(* PLC project SafeLOGIC, BrAutomation SafeDESIGNER  5.24.1.0 *)
(* stored: companyURL http://www.br-automation.com, creationDateTime Sun Oct 26 13:09:37 2025 *)

PROGRAM HeatWater

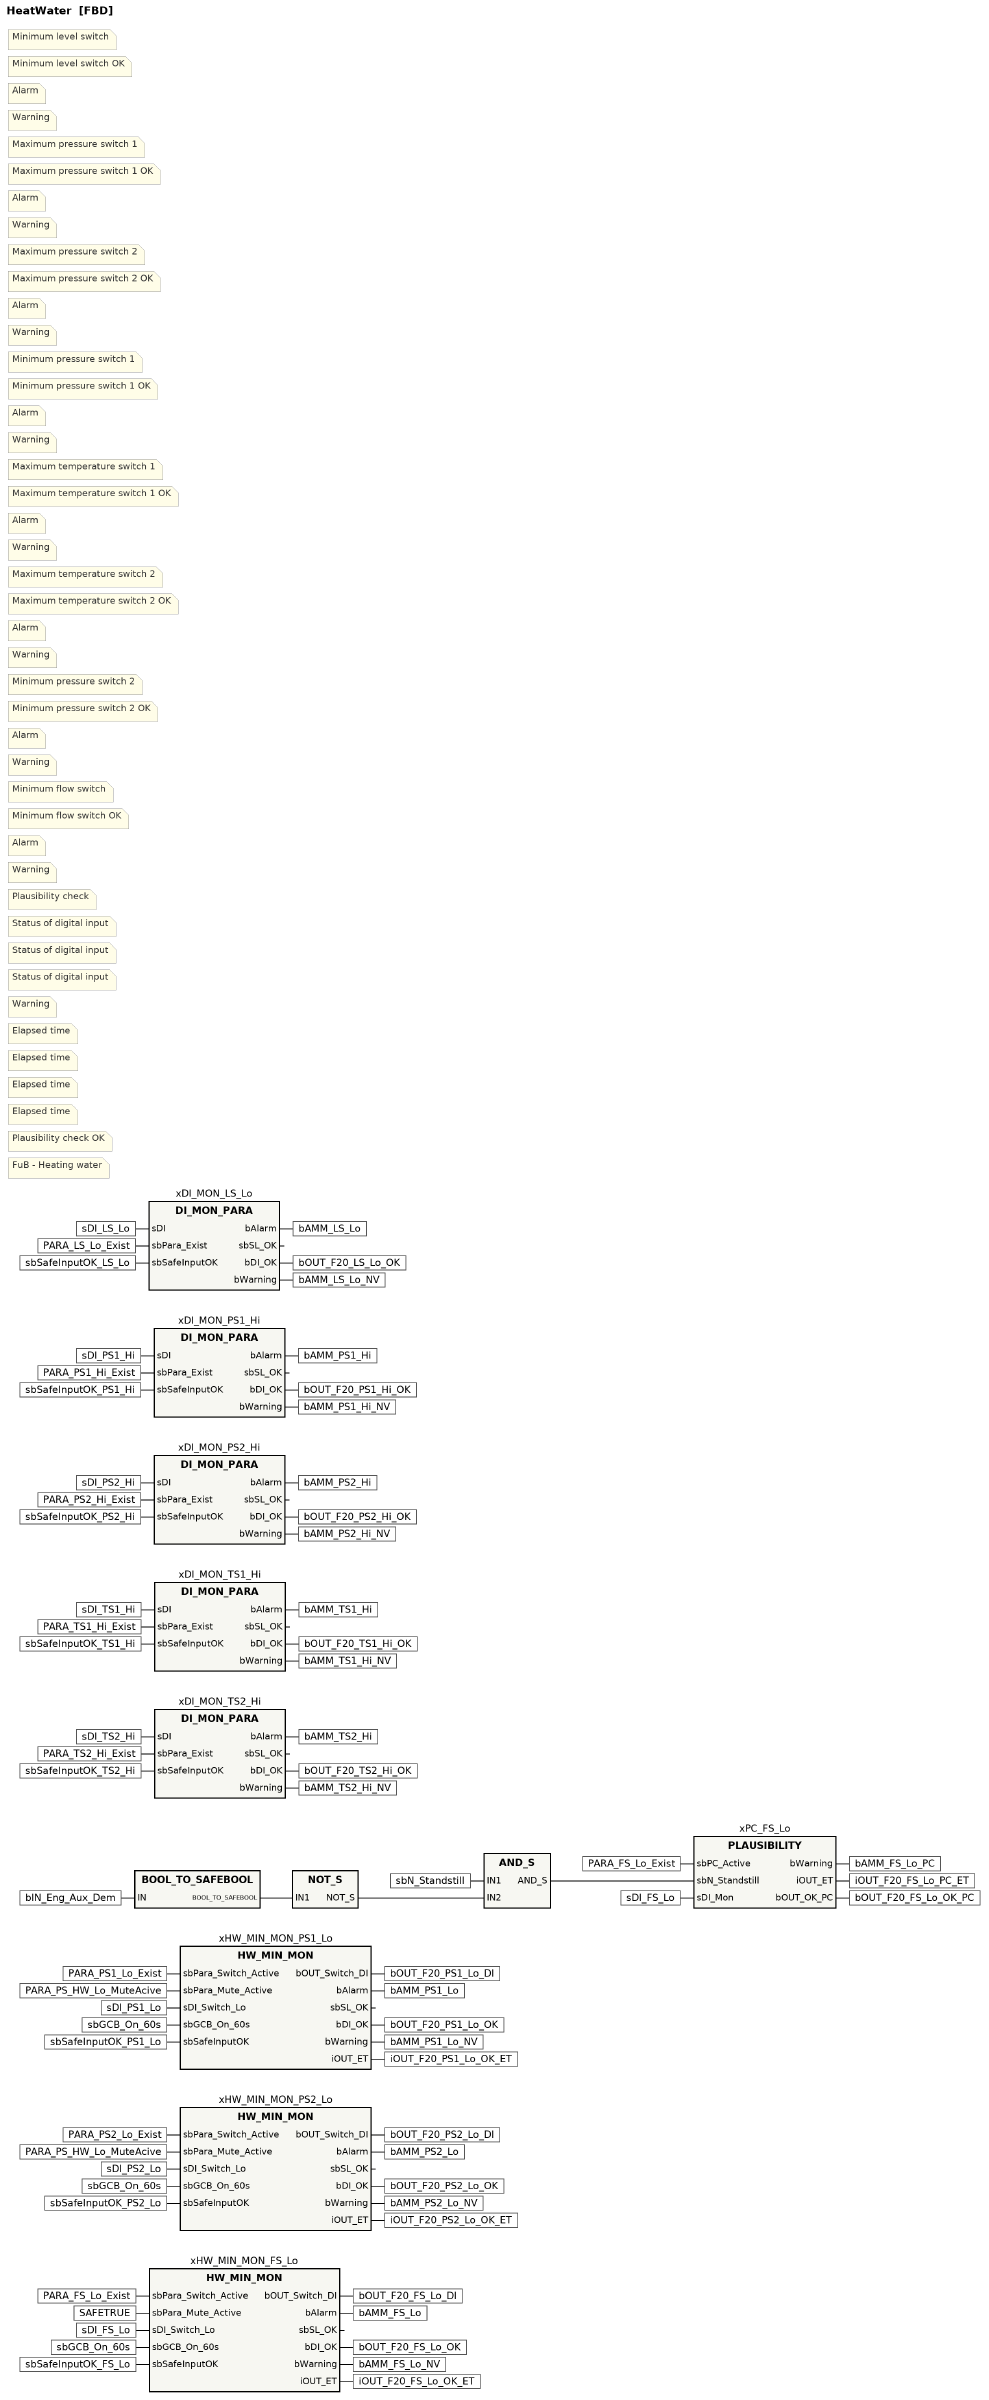
(* FBD diagram, written out as Structured Text *)
(* FuB - Heating water *)
(* Minimum level switch *)
(* Alarm *)
xDI_MON_LS_Lo(sDI := sDI_LS_Lo, sbPara_Exist := PARA_LS_Lo_Exist, sbSafeInputOK := sbSafeInputOK_LS_Lo);
bAMM_LS_Lo := xDI_MON_LS_Lo.bAlarm;
(* Minimum level switch OK *)
(* Warning *)
bAMM_LS_Lo_NV := xDI_MON_LS_Lo.bWarning;
bOUT_F20_LS_Lo_OK := xDI_MON_LS_Lo.bDI_OK;
(* Maximum pressure switch 1 *)
(* Alarm *)
xDI_MON_PS1_Hi(sDI := sDI_PS1_Hi, sbPara_Exist := PARA_PS1_Hi_Exist, sbSafeInputOK := sbSafeInputOK_PS1_Hi);
bAMM_PS1_Hi := xDI_MON_PS1_Hi.bAlarm;
(* Maximum pressure switch 1 OK *)
(* Warning *)
bAMM_PS1_Hi_NV := xDI_MON_PS1_Hi.bWarning;
bOUT_F20_PS1_Hi_OK := xDI_MON_PS1_Hi.bDI_OK;
(* Maximum pressure switch 2 *)
(* Alarm *)
xDI_MON_PS2_Hi(sDI := sDI_PS2_Hi, sbPara_Exist := PARA_PS2_Hi_Exist, sbSafeInputOK := sbSafeInputOK_PS2_Hi);
bAMM_PS2_Hi := xDI_MON_PS2_Hi.bAlarm;
(* Maximum pressure switch 2 OK *)
(* Warning *)
bAMM_PS2_Hi_NV := xDI_MON_PS2_Hi.bWarning;
bOUT_F20_PS2_Hi_OK := xDI_MON_PS2_Hi.bDI_OK;
(* Minimum pressure switch 1 *)
(* Status of digital input *)
(* Alarm *)
xHW_MIN_MON_PS1_Lo(sbPara_Switch_Active := PARA_PS1_Lo_Exist, sbPara_Mute_Active := PARA_PS_HW_Lo_MuteAcive, sDI_Switch_Lo := sDI_PS1_Lo, sbGCB_On_60s := sbGCB_On_60s, sbSafeInputOK := sbSafeInputOK_PS1_Lo);
bAMM_PS1_Lo := xHW_MIN_MON_PS1_Lo.bAlarm;
bOUT_F20_PS1_Lo_DI := xHW_MIN_MON_PS1_Lo.bOUT_Switch_DI;
(* Minimum pressure switch 1 OK *)
(* Warning *)
(* Elapsed time *)
bAMM_PS1_Lo_NV := xHW_MIN_MON_PS1_Lo.bWarning;
bOUT_F20_PS1_Lo_OK := xHW_MIN_MON_PS1_Lo.bDI_OK;
iOUT_F20_PS1_Lo_OK_ET := xHW_MIN_MON_PS1_Lo.iOUT_ET;
(* Minimum pressure switch 2 *)
(* Status of digital input *)
(* Alarm *)
xHW_MIN_MON_PS2_Lo(sbPara_Switch_Active := PARA_PS2_Lo_Exist, sbPara_Mute_Active := PARA_PS_HW_Lo_MuteAcive, sDI_Switch_Lo := sDI_PS2_Lo, sbGCB_On_60s := sbGCB_On_60s, sbSafeInputOK := sbSafeInputOK_PS2_Lo);
bAMM_PS2_Lo := xHW_MIN_MON_PS2_Lo.bAlarm;
bOUT_F20_PS2_Lo_DI := xHW_MIN_MON_PS2_Lo.bOUT_Switch_DI;
(* Minimum pressure switch 2 OK *)
(* Warning *)
(* Elapsed time *)
iOUT_F20_PS2_Lo_OK_ET := xHW_MIN_MON_PS2_Lo.iOUT_ET;
bAMM_PS2_Lo_NV := xHW_MIN_MON_PS2_Lo.bWarning;
bOUT_F20_PS2_Lo_OK := xHW_MIN_MON_PS2_Lo.bDI_OK;
(* Maximum temperature switch 1 *)
(* Alarm *)
xDI_MON_TS1_Hi(sDI := sDI_TS1_Hi, sbPara_Exist := PARA_TS1_Hi_Exist, sbSafeInputOK := sbSafeInputOK_TS1_Hi);
bAMM_TS1_Hi := xDI_MON_TS1_Hi.bAlarm;
(* Maximum temperature switch 1 OK *)
(* Warning *)
bAMM_TS1_Hi_NV := xDI_MON_TS1_Hi.bWarning;
bOUT_F20_TS1_Hi_OK := xDI_MON_TS1_Hi.bDI_OK;
(* Maximum temperature switch 2 *)
(* Alarm *)
xDI_MON_TS2_Hi(sDI := sDI_TS2_Hi, sbPara_Exist := PARA_TS2_Hi_Exist, sbSafeInputOK := sbSafeInputOK_TS2_Hi);
bAMM_TS2_Hi := xDI_MON_TS2_Hi.bAlarm;
(* Maximum temperature switch 2 OK *)
(* Warning *)
bAMM_TS2_Hi_NV := xDI_MON_TS2_Hi.bWarning;
bOUT_F20_TS2_Hi_OK := xDI_MON_TS2_Hi.bDI_OK;
(* Minimum flow switch *)
(* Status of digital input *)
(* Alarm *)
xHW_MIN_MON_FS_Lo(sbPara_Switch_Active := PARA_FS_Lo_Exist, sbPara_Mute_Active := SAFETRUE, sDI_Switch_Lo := sDI_FS_Lo, sbGCB_On_60s := sbGCB_On_60s, sbSafeInputOK := sbSafeInputOK_FS_Lo);
bAMM_FS_Lo := xHW_MIN_MON_FS_Lo.bAlarm;
bOUT_F20_FS_Lo_DI := xHW_MIN_MON_FS_Lo.bOUT_Switch_DI;
(* Minimum flow switch OK *)
(* Warning *)
(* Elapsed time *)
bAMM_FS_Lo_NV := xHW_MIN_MON_FS_Lo.bWarning;
bOUT_F20_FS_Lo_OK := xHW_MIN_MON_FS_Lo.bDI_OK;
iOUT_F20_FS_Lo_OK_ET := xHW_MIN_MON_FS_Lo.iOUT_ET;
(* Plausibility check *)
(* Warning *)
(* Elapsed time *)
(* Plausibility check OK *)
xPC_FS_Lo(sbPC_Active := PARA_FS_Lo_Exist, sbN_Standstill := AND_S(sbN_Standstill, NOT_S(BOOL_TO_SAFEBOOL(bIN_Eng_Aux_Dem))), sDI_Mon := sDI_FS_Lo);
iOUT_F20_FS_Lo_PC_ET := xPC_FS_Lo.iOUT_ET;
bAMM_FS_Lo_PC := xPC_FS_Lo.bWarning;
bOUT_F20_FS_Lo_OK_PC := xPC_FS_Lo.bOUT_OK_PC;
END_PROGRAM
